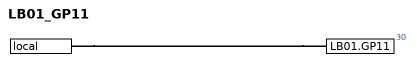
local := LB01.GP11;
ackLal S= local.ACK AND local.LAL;
ackHal S= local.ACK AND local.HAL;
local.ACK R= true;
// Alarm Low
local.CSP1 := local.SP - local.ADL;
gt_Min(IN := local.PV < local.CSP1 AND NOT SYS_StartupDelayComm AND LB01.GeneralStart AND LB01.TF1.Operating, PT := DINT_TO_TIME(local.AD * 60000)); // TON
AlarmAcknowledge01(Alarm := gt_Min.Q, InitPulse := SYS_InitPulse, AlarmAck := ackLal); // _BE_AlarmAckRemote
local.LAL := AlarmAcknowledge01.AlarmActive;
// Alarm High
local.CSP2 := local.SP + local.ADL;
gt_Max(IN := local.PV > local.CSP2 AND NOT SYS_StartupDelayComm AND LB01.GeneralStart AND LB01.TF1.Operating, PT := DINT_TO_TIME(local.AD * 60000)); // TON
AlarmAcknowledge02(Alarm := gt_Max.Q, InitPulse := SYS_InitPulse, AlarmAck := ackHal); // _BE_AlarmAckRemote
local.HAL := AlarmAcknowledge02.AlarmActive;
// Status HMI
IF true THEN _w1 := 0; END_IF
local.Symbol := _w1;
_w2 := local.LAL OR local.HAL;
IF _w2 THEN _w3 := 2; END_IF
local.AL := _w2;
local.Symbol := _w3;
LB01.GP11 := local;

END_PROGRAM

// Device/AREA1/B001/LB01/Sensor/Pressure/GP21/LB01_GP21
PROGRAM LB01_GP21
VAR
	local:strSensor2_Regulator;
	gt_Min: TON;
	gt_Max: TON;
	reset_en: RS;
	ackLal: BOOL;
	ackHal: BOOL;
	AlarmAcknowledge01: _BE_AlarmAckRemote;
	AlarmAcknowledge02: _BE_AlarmAckRemote;
END_VAR
VAR // added by the converter: edge detectors and wires of the graphical bodies
    _w1, _w3 : ANY;
    _w2 : BOOL;
END_VAR

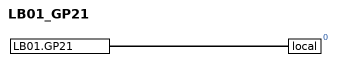
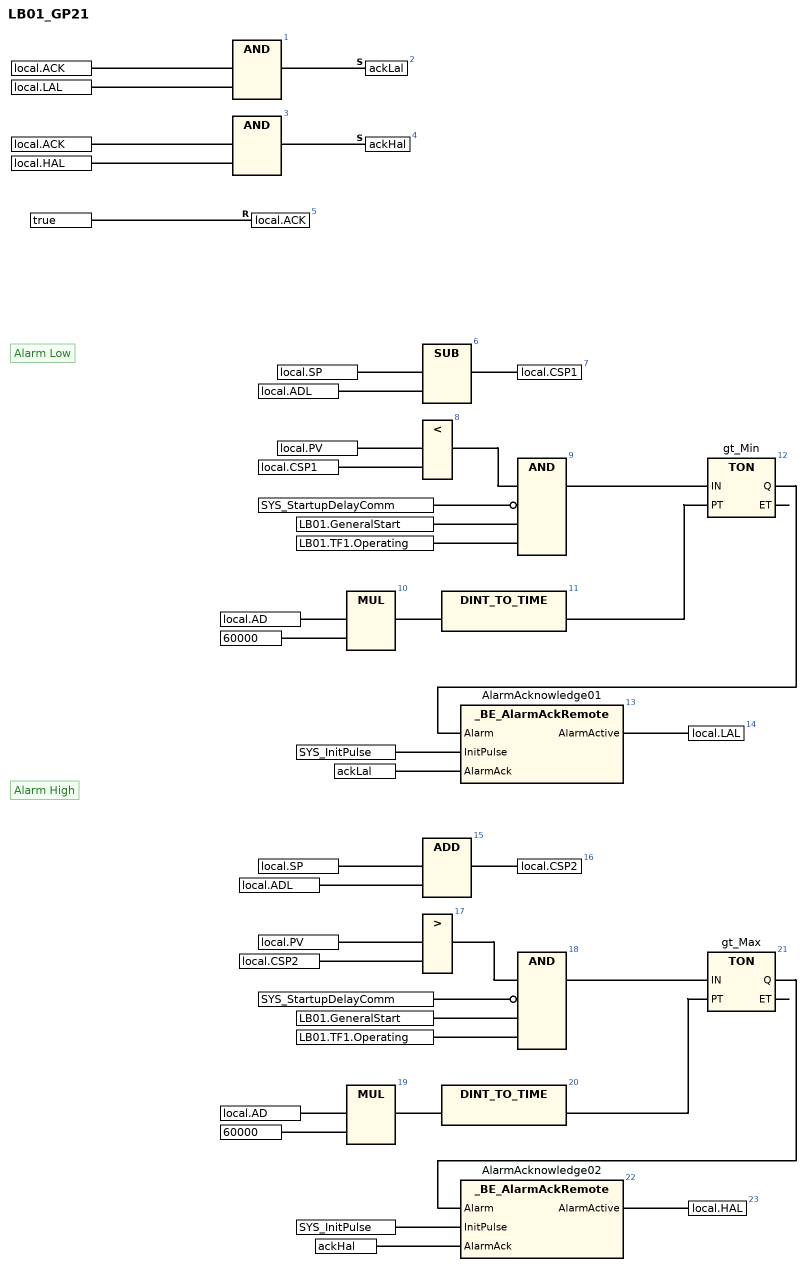
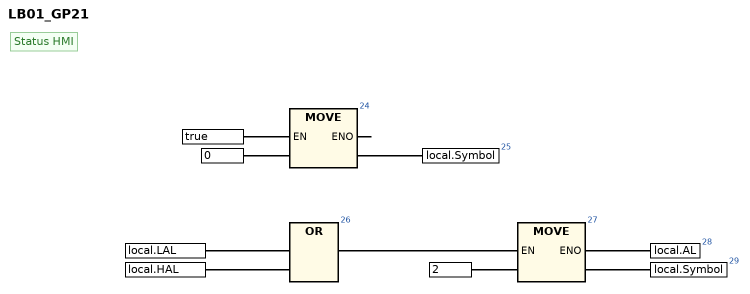
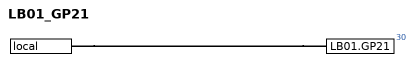
local := LB01.GP21;
ackLal S= local.ACK AND local.LAL;
ackHal S= local.ACK AND local.HAL;
local.ACK R= true;
// Alarm Low
local.CSP1 := local.SP - local.ADL;
gt_Min(IN := local.PV < local.CSP1 AND NOT SYS_StartupDelayComm AND LB01.GeneralStart AND LB01.TF1.Operating, PT := DINT_TO_TIME(local.AD * 60000)); // TON
AlarmAcknowledge01(Alarm := gt_Min.Q, InitPulse := SYS_InitPulse, AlarmAck := ackLal); // _BE_AlarmAckRemote
local.LAL := AlarmAcknowledge01.AlarmActive;
// Alarm High
local.CSP2 := local.SP + local.ADL;
gt_Max(IN := local.PV > local.CSP2 AND NOT SYS_StartupDelayComm AND LB01.GeneralStart AND LB01.TF1.Operating, PT := DINT_TO_TIME(local.AD * 60000)); // TON
AlarmAcknowledge02(Alarm := gt_Max.Q, InitPulse := SYS_InitPulse, AlarmAck := ackHal); // _BE_AlarmAckRemote
local.HAL := AlarmAcknowledge02.AlarmActive;
// Status HMI
IF true THEN _w1 := 0; END_IF
local.Symbol := _w1;
_w2 := local.LAL OR local.HAL;
IF _w2 THEN _w3 := 2; END_IF
local.AL := _w2;
local.Symbol := _w3;
LB01.GP21 := local;

END_PROGRAM

// Device/AREA1/B001/LB01/Sensor/Pressure/GP13/LB01_GP13
PROGRAM LB01_GP13
VAR
	local:strSensor4_FanGuard;
	AlarmAcknowledge01: _BE_AlarmAckRequired;
	fanGuardError: BOOL;
END_VAR
VAR // added by the converter: edge detectors and wires of the graphical bodies
    _w1, _w3 : ANY;
    _w2 : BOOL;
END_VAR

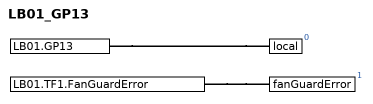
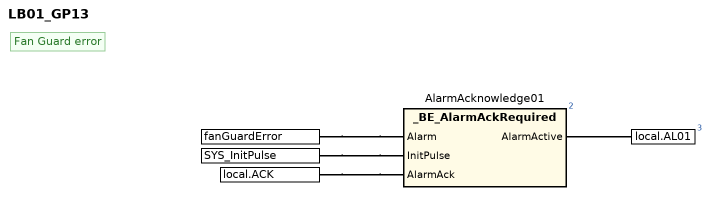
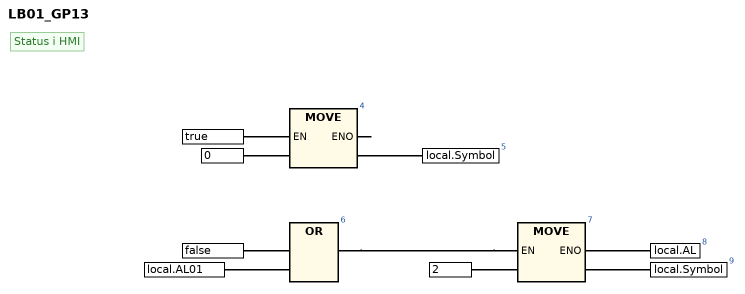
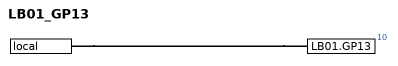
local := LB01.GP13;
fanGuardError := LB01.TF1.FanGuardError;
// Fan Guard error
AlarmAcknowledge01(Alarm := fanGuardError, InitPulse := SYS_InitPulse, AlarmAck := local.ACK); // _BE_AlarmAckRequired
local.AL01 := AlarmAcknowledge01.AlarmActive;
// Status i HMI
IF true THEN _w1 := 0; END_IF
local.Symbol := _w1;
_w2 := false OR local.AL01;
IF _w2 THEN _w3 := 2; END_IF
local.AL := _w2;
local.Symbol := _w3;
LB01.GP13 := local;

END_PROGRAM

// Device/AREA1/B001/LB01/Sensor/Pressure/GP23/LB01_GP23
PROGRAM LB01_GP23
VAR
	local:strSensor4_FanGuard;
	AlarmAcknowledge01: _BE_AlarmAckRequired;
	fanGuardError: BOOL;
END_VAR
VAR // added by the converter: edge detectors and wires of the graphical bodies
    _w1, _w3 : ANY;
    _w2 : BOOL;
END_VAR

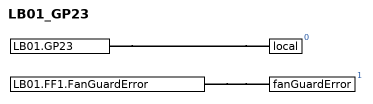
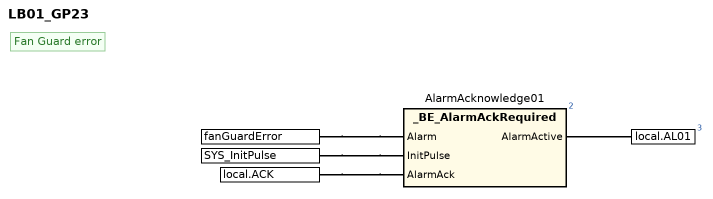
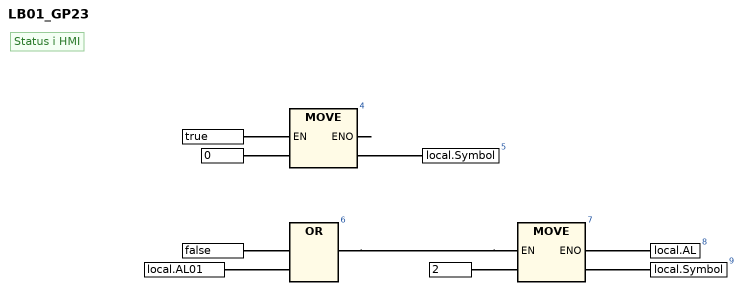
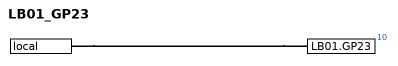
local := LB01.GP23;
fanGuardError := LB01.FF1.FanGuardError;
// Fan Guard error
AlarmAcknowledge01(Alarm := fanGuardError, InitPulse := SYS_InitPulse, AlarmAck := local.ACK); // _BE_AlarmAckRequired
local.AL01 := AlarmAcknowledge01.AlarmActive;
// Status i HMI
IF true THEN _w1 := 0; END_IF
local.Symbol := _w1;
_w2 := false OR local.AL01;
IF _w2 THEN _w3 := 2; END_IF
local.AL := _w2;
local.Symbol := _w3;
LB01.GP23 := local;

END_PROGRAM

// Device/AREA1/B001/LB01/Damper/ST11/LB01_ST11_Digital
PROGRAM LB01_ST11_Digital
VAR
	local:strDamper_Digital;
	FbPulse: R_TRIG;
	delayST11: TON;
	sp1: DINT;
	operating: BOOL;
	nh_v: BOOL;
END_VAR
VAR // added by the converter: edge detectors and wires of the graphical bodies
    _w1 : ANY;
END_VAR

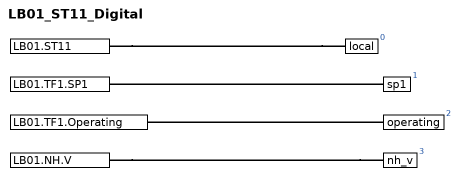
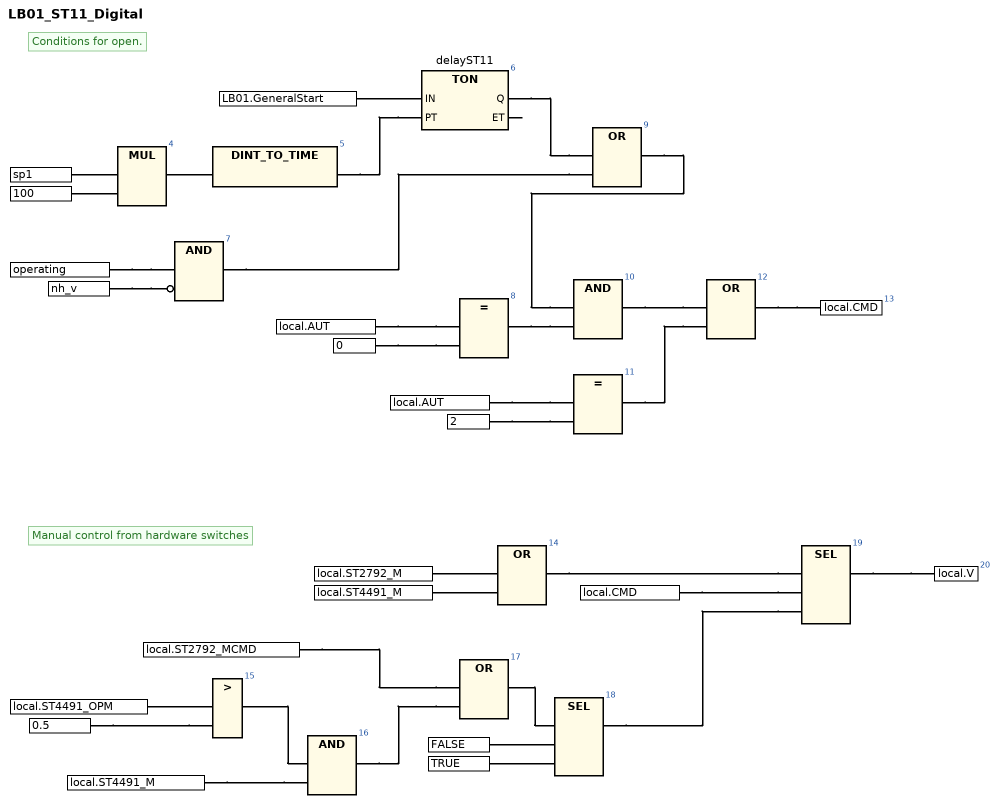
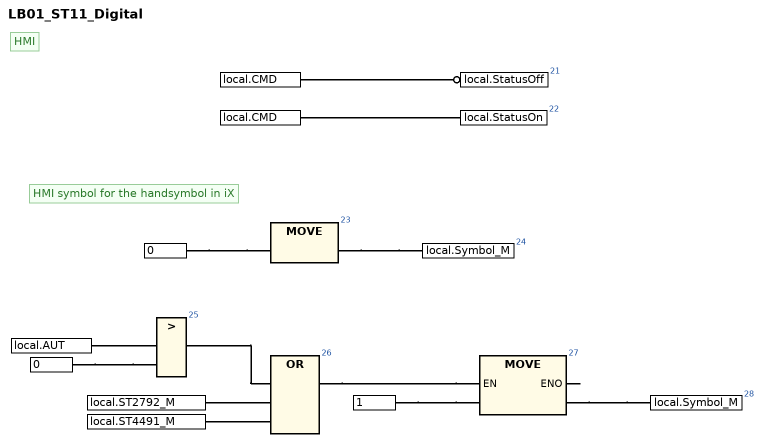
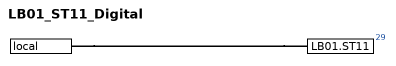
local := LB01.ST11;
sp1 := LB01.TF1.SP1;
operating := LB01.TF1.Operating;
nh_v := LB01.NH.V;
// Conditions for open.
delayST11(IN := LB01.GeneralStart, PT := DINT_TO_TIME(sp1 * 100)); // TON
local.CMD := (delayST11.Q OR operating AND NOT nh_v) AND local.AUT = 0 OR local.AUT = 2;
// Manual control from hardware switches
local.V := SEL(local.ST2792_M OR local.ST4491_M, local.CMD, SEL(local.ST2792_MCMD OR local.ST4491_OPM > 0.5 AND local.ST4491_M, FALSE, TRUE));
// HMI
local.StatusOff := NOT local.CMD;
local.StatusOn := local.CMD;
// HMI symbol for the handsymbol in iX
local.Symbol_M := 0;
IF local.AUT > 0 OR local.ST2792_M OR local.ST4491_M THEN _w1 := 1; END_IF
local.Symbol_M := _w1;
LB01.ST11 := local;

END_PROGRAM

// Device/AREA1/B001/LB01/Damper/ST21/LB01_ST21_Digital
PROGRAM LB01_ST21_Digital
VAR
	local:strDamper_Digital;
	FbPulse: R_TRIG;
	delayST11: TON;
	sp1: DINT;
	operating: BOOL;
	nh_v: BOOL;
END_VAR
VAR // added by the converter: edge detectors and wires of the graphical bodies
    _w1 : ANY;
END_VAR

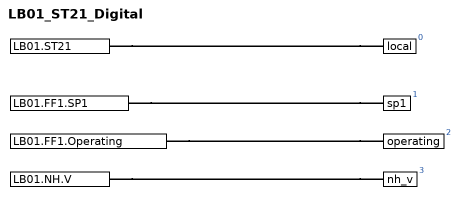
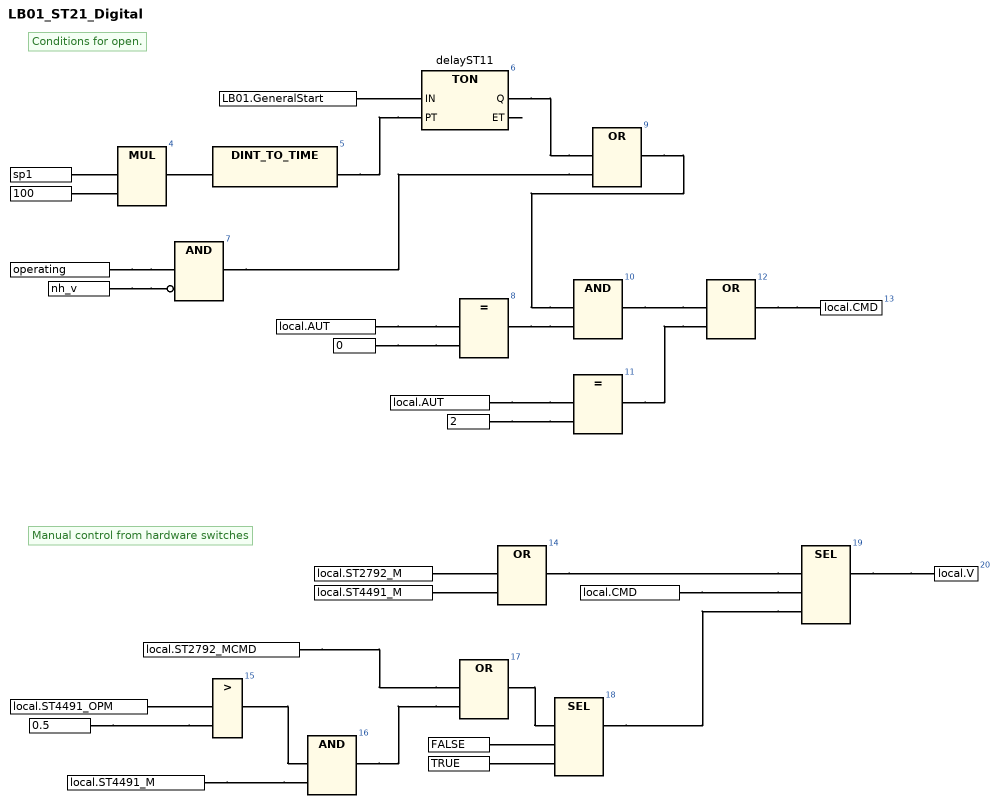
